(* CODESYS project Gates.project

Project tree, tasks and I/O mapping:
  Device : CODESYS Control Win V3, 3S - Smart Software Solutions GmbH, version 3.5.12.10
    application Application
      libraries: Standard, * (System)
      task MainTask (cyclic, interval t#20ms, priority 1) calls PLC_PRG
      task VISU_TASK (cyclic, interval 100 ms, priority 31) calls VisuElems.Visu_Prg
      program PLC_PRG [LD]
      visualisation Visualization
  text list GlobalTextList
*)

// Device/Application/PLC_PRG
PROGRAM PLC_PRG
VAR
	Input1: BOOL;
	Input2: BOOL;
	Lamp1: BOOL;
END_VAR

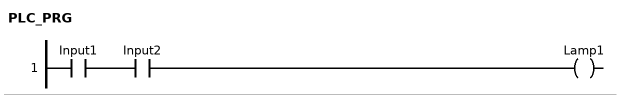
// NETWORK 1
Lamp1 := Input1 AND Input2;

END_PROGRAM

// Device/Application/Visualization
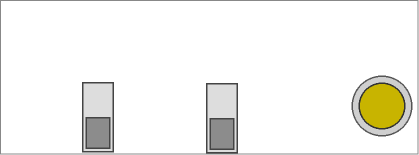
VISUALIZATION Visualization  // 419x155
    Lamp1 (347,71 70x70), variable: PLC_PRG.Lamp1, style: Lamp-Lamp1-Yellow
    DipSwitch (63,82 70x70), variable: PLC_PRG.Input1, behaviour: TOGGLE, style: Switch-DipSwitch-Gray
    DipSwitch (187,83 70x70), variable: PLC_PRG.Input2, behaviour: TOGGLE, style: Switch-DipSwitch-Gray
END_VISUALIZATION
